KUKA KRL program: inline_arc_fn.src, inline_arc_fn.dat

--- inline_arc_fn.src ---
&ACCESS RV
&REL 5
&COMMENT try with dat
&PARAM EDITMASK = *
&PARAM TEMPLATE = C:\KRC\Roboter\Template\vorgabe
&PARAM DISKPATH = KRC:\R1
DEF inline_arc_fn( )
;()1234 5678
END


GLOBAL DEF INLINE_ARC_ON(gcode_cmd :IN)
   DECL GCODE_CMD_T gcode_cmd
   DECL INT job_number ; this is the emission intensity

   ; Cast emission float to integer job number
   job_number = gcode_cmd.E

   ; the job numbers are set up such that job 1 is one CMT droplet, job 2 .. two CMT droplets
   ; therefore the job number is a proxy to the Emission intensity



   JOB_WELD_DAT.Weld.Channel1 = job_number ; Update the specific variable
   ; whenever we start the weld job we start on channel 1
  ;  JOB_WELD_DAT.Weld.Channel1 = 1

   ; as far as i understand CD_PARAMS is for the torque based collision detection on the axis.
  ;  SET_CD_PARAMS (2) ;

     ; in our case colision detect is happening on $IN[9] - the fronius crashbox
     ; managed by `sps.sub` ArcTech loop

   TRIGGER WHEN DISTANCE = 1 DELAY = ArcGetDelay(#PreDefinition, JOB_WELD_DAT) DO ArcMainNG(#PreDefinition, JOB_WELD_DAT, CP_DAT_VESTIGIAL) PRIO = -1
   TRIGGER WHEN PATH = ArcGetPath(#OnTheFlyArcOn, JOB_WELD_DAT) DELAY = ArcGetDelay(#GasPreflow, JOB_WELD_DAT) DO ArcMainNG(#GasPreflow, JOB_WELD_DAT, CP_DAT_VESTIGIAL) PRIO = -1
   TRIGGER WHEN PATH = ArcGetPath(#OnTheFlyArcOn, JOB_WELD_DAT) DELAY = ArcGetDelay(#ArcPreOn, JOB_WELD_DAT) DO ArcMainNG(#ArcOnMoveStd, JOB_WELD_DAT, CP_DAT_VESTIGIAL) PRIO = -1
   ArcMainNG(#ArcOnBeforeMoveStd, JOB_WELD_DAT, CP_DAT_VESTIGIAL)
   LIN_safe(gcode_cmd)
   ArcMainNG(#ArcOnAfterMoveStd, JOB_WELD_DAT, CP_DAT_VESTIGIAL)

;FOLD ARCON JOB_WELD_DAT LIN gotoPt Vel=0.02 m/s CPDAT1 Tool[5]:nx_mtb500_10mm Base[0] ;%{PE}
;FOLD Parameters ;%{h}
;Params IlfProvider=kukaroboter.arctech.arconlin; Kuka.IsGlobalPoint=False; Kuka.PointName=gotoPt; Kuka.BlendingEnabled=False; Kuka.MoveDataName=CPDAT1; Kuka.VelocityPath=0.02; Kuka.CurrentCDSetIndex=0; Kuka.MovementParameterFieldEnabled=True; ArcTech.WdatVarName=JOB_WELD_DAT; ArcTech.Basic=3.6.2.371
;ENDFOLD
;$BWDSTART = FALSE
;LDAT_ACT = LCPDAT1
;FDAT_ACT = FgotoPt
;BAS(#CP_PARAMS, 0.02)
;SET_CD_PARAMS (0)
;TRIGGER WHEN DISTANCE = 1 DELAY = ArcGetDelay(#PreDefinition, JOB_WELD_DAT) DO ArcMainNG(#PreDefinition, JOB_WELD_DAT, CP_DAT_VESTIGIAL) PRIO = -1
;TRIGGER WHEN PATH = ArcGetPath(#OnTheFlyArcOn, JOB_WELD_DAT) DELAY = ArcGetDelay(#GasPreflow, JOB_WELD_DAT) DO ArcMainNG(#GasPreflow, JOB_WELD_DAT, CP_DAT_VESTIGIAL) PRIO = -1
;TRIGGER WHEN PATH = ArcGetPath(#OnTheFlyArcOn, JOB_WELD_DAT) DELAY = ArcGetDelay(#ArcPreOn, JOB_WELD_DAT) DO ArcMainNG(#ArcOnMoveStd, JOB_WELD_DAT, CP_DAT_VESTIGIAL) PRIO = -1
;ArcMainNG(#ArcOnBeforeMoveStd, JOB_WELD_DAT, CP_DAT_VESTIGIAL)
;LIN g1_pos C_VEL
;ArcMainNG(#ArcOnAfterMoveStd, JOB_WELD_DAT, CP_DAT_VESTIGIAL)
;ENDFOLD
;FOLD INI;%{PE}
  ;FOLD BASISTECH INI
;;;    GLOBAL INTERRUPT DECL 3 WHEN $STOPMESS==TRUE DO IR_STOPM ( )
;;;    INTERRUPT ON 3
;;;    BAS (#INITMOV,0 )
  ;ENDFOLD (BASISTECH INI)
  ;FOLD USER INI
    ;Make your modifications here

  ;ENDFOLD (USER INI)
;ENDFOLD (INI)

;FOLD SPTP HOME Vel=100 % DEFAULT ;%{PE}
;FOLD Parameters ;%{h}
;Params IlfProvider=kukaroboter.basistech.inlineforms.movement.spline; Kuka.IsGlobalPoint=False; Kuka.PointName=HOME; Kuka.BlendingEnabled=False; Kuka.MoveDataPtpName=DEFAULT; Kuka.VelocityPtp=100; Kuka.VelocityFieldEnabled=True; Kuka.CurrentCDSetIndex=0; Kuka.MovementParameterFieldEnabled=True; IlfCommand=SPTP
;ENDFOLD
;;;SPTP XHOME WITH $VEL_AXIS[1] = SVEL_JOINT(100.0), $TOOL = STOOL2(FHOME), $BASE = SBASE(FHOME.BASE_NO), $IPO_MODE = SIPO_MODE(FHOME.IPO_FRAME), $LOAD = SLOAD(FHOME.TOOL_NO), $ACC_AXIS[1] = SACC_JOINT(PDEFAULT), $APO = SAPO_PTP(PDEFAULT), $GEAR_JERK[1] = SGEAR_JERK(PDEFAULT), $COLLMON_TOL_PRO[1] = USE_CM_PRO_VALUES(0)
;ENDFOLD

;FOLD SPTP HOME Vel=100 % DEFAULT ;%{PE}
;FOLD Parameters ;%{h}
;Params IlfProvider=kukaroboter.basistech.inlineforms.movement.spline; Kuka.IsGlobalPoint=False; Kuka.PointName=HOME; Kuka.BlendingEnabled=False; Kuka.MoveDataPtpName=DEFAULT; Kuka.VelocityPtp=100; Kuka.VelocityFieldEnabled=True; Kuka.CurrentCDSetIndex=0; Kuka.MovementParameterFieldEnabled=True; IlfCommand=SPTP
;ENDFOLD
;;;SPTP XHOME WITH $VEL_AXIS[1] = SVEL_JOINT(100.0), $TOOL = STOOL2(FHOME), $BASE = SBASE(FHOME.BASE_NO), $IPO_MODE = SIPO_MODE(FHOME.IPO_FRAME), $LOAD = SLOAD(FHOME.TOOL_NO), $ACC_AXIS[1] = SACC_JOINT(PDEFAULT), $APO = SAPO_PTP(PDEFAULT), $GEAR_JERK[1] = SGEAR_JERK(PDEFAULT), $COLLMON_TOL_PRO[1] = USE_CM_PRO_VALUES(0)
;ENDFOLD


END

GLOBAL DEF INLINE_ARC_SWI(gcode_cmd :IN)
   DECL GCODE_CMD_T gcode_cmd
   DECL INT job_number ; this is the emission intensity

   ; Cast emission float to integer job number
   job_number = gcode_cmd.E

   ; the job numbers are set up such that job 1 is one CMT droplet, job 2 .. two CMT droplets
   ; therefore the job number is a proxy to the Emission intensity



   JOB_WELD_DAT.Weld.Channel1 = job_number ; Update the specific variable


;FOLD ARCSWI <JOB_WELD_DAT> LIN gotoPt CPDAT2 Tool[5]:nx_mtb500_10mm Base[0] ColDetect[9] ;%{PE}
;FOLD Parameters ;%{h}
;Params IlfProvider=kukaroboter.arctech.arcswilin; Kuka.IsGlobalPoint=False; Kuka.PointName=gotoPt; Kuka.BlendingEnabled=True; Kuka.MoveDataName=CPDAT2; Kuka.VelocityPath=0.02; Kuka.CurrentCDSetIndex=9; Kuka.MovementParameterFieldEnabled=True; ArcTech.Global.WdatVarName=gJOB_WELD_DAT; ArcTech.IsGlobalWdat=True; ArcTech.Basic=3.6.2.371
;ENDFOLD
;$BWDSTART = FALSE
;LDAT_ACT = LCPDAT2
;FDAT_ACT = FgotoPt
;BAS(#CP_PARAMS, gArcBasVelDefinition)
; SET_CD_PARAMS (9)


TRIGGER WHEN DISTANCE = 1 DELAY = 0 DO ArcMainNG(#ArcSwiMoveStd, JOB_WELD_DAT, CP_DAT_VESTIGIAL) PRIO = -1
ArcMainNG(#ArcSwiBeforeMoveStd, JOB_WELD_DAT, CP_DAT_VESTIGIAL)
; LIN g1_pos C_VEL
LIN_safe(gcode_cmd)
ArcMainNG(#ArcSwiAfterMoveStd, JOB_WELD_DAT, CP_DAT_VESTIGIAL)
;ENDFOLD
END

GLOBAL DEF INLINE_ARC_STOP(gcode_cmd :IN)
   DECL GCODE_CMD_T gcode_cmd



; SET_CD_PARAMS (9)
TRIGGER WHEN PATH = ArcGetPath(#ArcOffBefore, JOB_WELD_DAT) DELAY = 0 DO ArcMainNG(#ArcOffBeforeOffStd, JOB_WELD_DAT, CP_DAT_VESTIGIAL) PRIO = -1
TRIGGER WHEN PATH = ArcGetPath(#ArcOffBefore2, JOB_WELD_DAT) DELAY = 0 DO ArcMainNG(#ArcOffBeforeOffStd2, JOB_WELD_DAT, CP_DAT_VESTIGIAL) PRIO = -1
TRIGGER WHEN PATH = ArcGetPath(#OnTheFlyArcOff, JOB_WELD_DAT) DELAY = 0 DO ArcMainNG(#ArcOffMoveStd, JOB_WELD_DAT, CP_DAT_VESTIGIAL) PRIO = -1
ArcMainNG(#ArcOffBeforeMoveStd, JOB_WELD_DAT, CP_DAT_VESTIGIAL)
LIN_safe(gcode_cmd)
ArcMainNG(#ArcOffAfterMoveStd, JOB_WELD_DAT, CP_DAT_VESTIGIAL)


;FOLD ARCOFF <G_WDAT> LIN G_PT CPDAT3 Tool[5]:nx_mtb500_10mm Base[0] ColDetect[9] ;%{PE}
;FOLD Parameters ;%{h}
;Params IlfProvider=kukaroboter.arctech.arcofflin; Kuka.IsGlobalPoint=False; Kuka.PointName=G_PT; Kuka.BlendingEnabled=False; Kuka.MoveDataName=CPDAT3; Kuka.VelocityPath=0.02; Kuka.CurrentCDSetIndex=9; Kuka.MovementParameterFieldEnabled=True; ArcTech.Global.WdatVarName=gG_WDAT; ArcTech.IsGlobalWdat=True; ArcTech.Basic=3.6.2.371
;ENDFOLD

;ENDFOLD
END

--- inline_arc_fn.dat ---
&ACCESS RV1
&REL 4
&COMMENT try with dat
&PARAM EDITMASK = *
&PARAM TEMPLATE = C:\KRC\Roboter\Template\vorgabe
&PARAM DISKPATH = KRC:\R1
DEFDAT  INLINE_ARC_FN
;()12345555 567
EXT  BAS (BAS_COMMAND  :IN,REAL  :IN )
DECL INT SUCCESS

DECL stArcDat_T JOB_WELD_DAT={WdatId[] "ARC_ON_WELD_DAT",Info {Version 306020371,WId 1,WName[] "Fronius TPSi job mode"},Strike {JobModeId[] "Job mode",StartTime 0.0,PreFlowTime 0.0,Channel1 0.0,Channel2 0.0,Channel3 0.0,Channel4 0.0,Channel5 0.0,Channel6 0.0,Channel7 0.0,Channel8 0.0,PurgeTime 0.0},Weld {JobModeId[] "Job mode",ParamSetId[] "Set1",Velocity 0.00250000,Channel1 2.00000,Channel2 0.0,Channel3 0.0,Channel4 0.0,Channel5 0.0,Channel6 0.0,Channel7 0.0,Channel8 0.0},Weave {Pattern #None,Length 4.00000,Amplitude 2.00000,Angle 0.0,Frequency 2.00000,LeftSideDelay 0.0,RightSideDelay 0.0}}

; this is the motion dataset .. it is not used for anything because we manage motion externally.
DECL stArcDat_T CP_DAT_VESTIGIAL={WdatId[] "WCP_POINT_DATA",Info {Version 306020371},Strike {SeamName[] "seamsAbitFishy",PartName[] "waamapart",SeamNumber 1,PartNumber 1,DesiredLength 1.00000,LengthTolNeg 0.0,LengthTolPos 0.0,LengthCtrlActive FALSE},Advanced {BitCodedRobotMark 0}}




; DECL stArcDat_T ARC_ON_WELD_DAT={WdatId[] "ARC_ON_WELD_DAT",Info {Version 306020371,WId 1,WName[] "Fronius TPSi job mode"},Strike {JobModeId[] "Job mode",StartTime 0.0,PreFlowTime 0.0,Channel1 0.0,Channel2 0.0,Channel3 0.0,Channel4 0.0,Channel5 0.0,Channel6 0.0,Channel7 0.0,Channel8 0.0,PurgeTime 0.0},Weld {JobModeId[] "Job mode",ParamSetId[] "Set1",Velocity 0.00250000,Channel1 2.00000,Channel2 0.0,Channel3 0.0,Channel4 0.0,Channel5 0.0,Channel6 0.0,Channel7 0.0,Channel8 0.0},Weave {Pattern #None,Length 4.00000,Amplitude 2.00000,Angle 0.0,Frequency 2.00000,LeftSideDelay 0.0,RightSideDelay 0.0}}

; DECL stArcDat_T WCP_POINT_DATA={WdatId[] "WCP_POINT_DATA",Info {Version 306020371},Strike {SeamName[] "seamsAbitFishy",PartName[] "waamapart",SeamNumber 1,PartNumber 1,DesiredLength 1.00000,LengthTolNeg 0.0,LengthTolPos 0.0,LengthCtrlActive FALSE},Advanced {BitCodedRobotMark 0}}

; DECL E6POS XCP_POINT_DATA={X 1800.00037,Y 60.0004158,Z 1699.99963,A -92.2002792,B -0.576508343,C 0.250116497,S 18,T 35,E1 0.0,E2 0.0,E3 0.0,E4 0.0,E5 0.0,E6 0.0}
; DECL FDAT FCP_POINT_DATA={TOOL_NO 5,BASE_NO 0,IPO_FRAME #BASE,POINT2[] " "}
; DECL LDAT LCPDAT2={VEL 0.0200000,ACC 100.000,APO_DIST 500.000,APO_FAC 50.0000,AXIS_VEL 100.000,AXIS_ACC 100.000,ORI_TYP #VAR,CIRC_TYP #BASE,JERK_FAC 50.0000,GEAR_JERK 100.000,EXAX_IGN 0,CB {AUX_PT {ORI #CONSIDER,E1 #CONSIDER,E2 #CONSIDER,E3 #CONSIDER,E4 #CONSIDER,E5 #CONSIDER,E6 #CONSIDER},TARGET_PT {ORI #INTERPOLATE,E1 #INTERPOLATE,E2 #INTERPOLATE,E3 #INTERPOLATE,E4 #INTERPOLATE,E5 #INTERPOLATE,E6 #INTERPOLATE}}}
; DECL MODULEPARAM_T LAST_TP_PARAMS={PARAMS[] "Kuka.PointName=CP_POINT_DATA; Kuka.FrameData.base_no=0; Kuka.FrameData.tool_no=5; Kuka.FrameData.ipo_frame=#BASE; Kuka.isglobalpoint=False; Kuka.MoveDataName=CPDAT2; Kuka.MovementData.cb={AUX_PT {ORI #CONSIDER,E1 #CONSIDER,E2 #CONSIDER,E3 #CONSIDER,E4 #CONSIDER,E5 #CONSIDER,E6 #CONSIDER},TARGET_PT {ORI #INTERPOLATE,E1 #INTERPOLATE,E2 #INTERPOLATE,E3 #INTERPOLATE,E4 #INTERPOLATE,E5 #INTERPOLATE,E6 #INTERPOLATE}}; Kuka.MovementData.apo_fac=50; Kuka.MovementData.apo_dist=500; Kuka.MovementData.axis_acc=100; Kuka.MovementData.axis_vel=100; Kuka.MovementData.circ_typ=#BASE; Kuka.MovementData.jerk_fac=50; Kuka.MovementData.ori_typ=#VAR; Kuka.MovementData.vel=0.02; Kuka.MovementData.acc=100; Kuka.MovementData.exax_ign=0; Kuka.VelocityPath=0.02; Kuka.BlendingEnabled=False; Kuka.APXEnabled=False; Kuka.CurrentCDSetIndex=1; ArcTech.WdatVarName=ARC_ON_WELD_DAT"}
ENDDAT
